{attribute 'GeneratedUsingTerminal: EP3752-0000-0017'}
{attribute addProperty BoxType "EP3752-0000-0017"}
{attribute addProperty Id "StatusAT %I*Status_8F1D55D83ValueAT %I*INT2"}
{attribute addProperty CRC "1518760301"}
{attribute addProperty Size "5"}
TYPE AI_Inputs_Channel_5A86716D :
STRUCT
	{attribute addProperty Name "Status"}
	Status AT %I* : Status_8F1D55D8;
	{attribute addProperty Name "Value"}
	Value AT %I* : INT;
END_STRUCT
END_TYPE

(* stored: Version 1.2.0.0, ProductVersion 3.1.4024.9
   DUT AI_Inputs_Channel_5A86716D: Id {9469839a-c70d-431c-9097-63b60988cb66} *)
